KUKA KRL data list: PolishInitialization.dat

&ACCESS RVP
&REL 105
&COMMENT Polish Init 250608
&PARAM DISKPATH = KRC:\R1\Program\SbtComm012Polish
DEFDAT  POLISHINITIALIZATION

DECL MODULEPARAM_T LAST_TP_PARAMS={PARAMS[] "SBTCOMM012.GRINDHEADID=4; SBTCOMM012.TOOLDATA=0; SBTCOMM012.SPINDLESPEED=6000; SBTCOMM012.TOOLDIRECTION=5; SBTCOMM012.GRINDENABLE=True; SBTCOMM012.DOUTINDEX=0; SBTCOMM012.DININDEX=0                                                  "}
ENDDAT
